# EPICS substitutions: ek9000App/Db/EL2794.substitutions
file EL2794.template
{       pattern
        {
                TERMINAL,

        }
        {
        }
}
